// TIA Portal V17 export
// export: Created 2025-03-10T13:12:45.1088536Z, ExportSetting WithDefaults, DisplayName Totally Integrated Automation Portal, DisplayVersion V17 Update 8, DisplayName TIA Portal Openness, DisplayVersion V17 Update 8, DisplayName TIA Portal Version Control Interface, DisplayVersion V17, DisplayName SINAMICS Startdrive Advanced, DisplayVersion V17 SP2, DisplayName SINAMICS Startdrive G110M, G120, G120C, G120D, G120P, G115D, DisplayVersion V17 SP2, DisplayName SINAMICS Startdrive G130, G150, S120, S150, SINAMICS MV, S210, DisplayVersion V17 SP2, DisplayName STEP 7 Professional, DisplayVersion V17 Update 8, DisplayName SINUMERIK ONE STEP 7 Toolbox, DisplayVersion V17 Update 12, DisplayName SINUMERIK 840D sl STEP 7 Toolbox, DisplayVersion V17 Update 12, DisplayName STEP 7 Safety, DisplayVersion V17 Update 6, DisplayName WinCC Advanced, DisplayVersion V17 Update 8
DATA_BLOCK "DB16703_OPC_UA_HOPPER_1_UNIT_01"   // DB16703
VERSION : 0.1
// stored: AutoNumber false, DBAccessibleFromOPCUA true, DBAccessibleFromWebserver true, InstanceOfName FB16702_OPC_UA_HOPPER_DATA, InstanceOfType FB
"FB16702_OPC_UA_HOPPER_DATA"
   // VAR_INPUT
   //    PRESSURIZE_GAS_VALVE { ExternalWritable := 'False'} : Bool;
   //    RELIEVE_GAS_VALVE { ExternalWritable := 'False'} : Bool;
   //    HIGH_LEVEL { ExternalWritable := 'False'} : Bool;
   //    LOW_LEVEL { ExternalWritable := 'False'} : Bool;
   //    MAX_WEIGHT_SETPOINT { ExternalWritable := 'False'} : Real;
   //    TOTAL_WEIGHT { ExternalWritable := 'False'} : Real;
   //    HOPPER_WEIGHT_SETPOINT { ExternalWritable := 'False'} : Real;
   //    POWDER_WEIGHT { ExternalWritable := 'False'} : Real;
   //    UPPER_JACKET_TEMPERATURE { ExternalWritable := 'False'} : Real;
   //    UPPER_JACKET_TEMPERATURE_SETPOINT { ExternalWritable := 'False'} : Real;
   //    LOWER_JACKET_TEMPERATURE { ExternalWritable := 'False'} : Real;
   //    LOWER_JACKET_TEMPERATURE_SETPOINT { ExternalWritable := 'False'} : Real;
   //    HOPPER_COVER { ExternalWritable := 'False'} : Real;
   //    HOPPER_COVER_SETPOINT { ExternalWritable := 'False'} : Real;
   //    STIRRER_CURRENT { ExternalWritable := 'False'} : DInt;
   //    STIRRER_SPEED { ExternalWritable := 'False'} : DInt;
   //    STIRRER_SPEED_SETPOINT { ExternalWritable := 'False'} : DInt;
   //    TRANSFER_POWDER_VALVE { ExternalWritable := 'False'} : Bool;
   //    CLEANING_AIR_VALVE { ExternalWritable := 'False'} : Bool;
   //    LOAD_FEEDER_SEQ { ExternalWritable := 'False'} : Bool;
   //    MEDICOAT_DATA : Int;
   // END_VAR
   // VAR_IN_OUT
   //    HOPPER : "HOPPER";
   // END_VAR
   // VAR
   //    POWDER_FLOW_DATA_SAVE { S7_SetPoint := 'True'} : "FB16700_POWDER_FLOW_DATA_SAVE";
   // END_VAR
BEGIN
END_DATA_BLOCK
